// SIMATIC S7-200 project (STEP 7-Micro/WIN), CPU 226 REL 01.23

ORGANIZATION_BLOCK 主程序:OB1
TITLE=
BEGIN
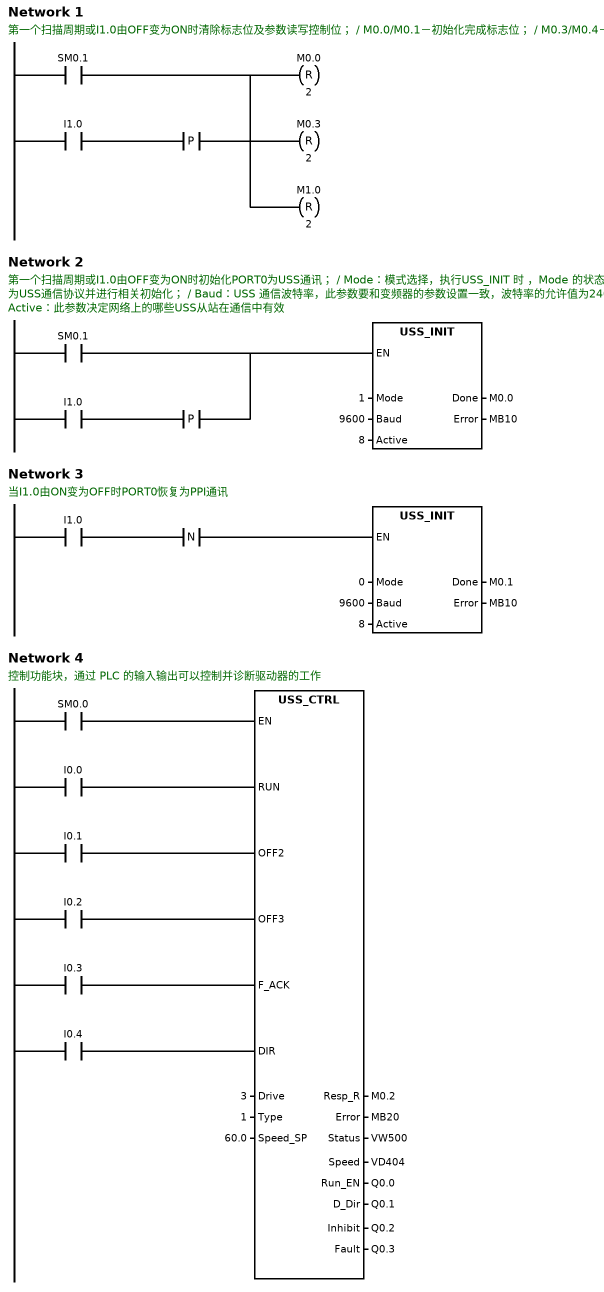
Network 1
// 第一个扫描周期或I1.0由OFF变为ON时清除标志位及参数读写控制位；
// M0.0/M0.1－初始化完成标志位；
// M0.3/M0.4－读写功能块完成标志位，用于功能块轮替；
// M1.0/M1.1－读写功能块控制位
LD     SM0.1
LD     I1.0
EU
OLD
R      M0.0, 2
R      M0.3, 2
R      M1.0, 2
Network 2
// 第一个扫描周期或I1.0由OFF变为ON时初始化PORT0为USS通讯；
// Mode：模式选择，执行USS_INIT 时 ，Mode 的状态决定 是否在Port上使用USS通信功能，0 - 恢复 Port 0 为PPI从站模式，1 - 设置 Port 0 为USS通信协议并进行相关初始化；
// Baud：USS 通信波特率，此参数要和变频器的参数设置一致，波特率的允许值为2400、4800、9600、19200、38400、57600 或115200 bit/s； 
// Active：此参数决定网络上的哪些USS从站在通信中有效
LD     SM0.1
LD     I1.0
EU
OLD
CALL   USS_INIT:SBR5, 1, 9600, 8, M0.0, MB10
Network 3
// 当I1.0由ON变为OFF时PORT0恢复为PPI通讯
LD     I1.0
ED
CALL   USS_INIT:SBR5, 0, 9600, 8, M0.1, MB10
Network 4
// 控制功能块，通过 PLC 的输入输出可以控制并诊断驱动器的工作
LD     SM0.0
=      L60.0
LD     I0.0
=      L63.7
LD     I0.1
=      L63.6
LD     I0.2
=      L63.5
LD     I0.3
=      L63.4
LD     I0.4
=      L63.3
LD     L60.0
CALL   USS_CTRL:SBR2, L63.7, L63.6, L63.5, L63.4, L63.3, 3, 1, 60.0, M0.2, MB20, VW500, VD404, Q0.0, Q0.1, Q0.2, Q0.3
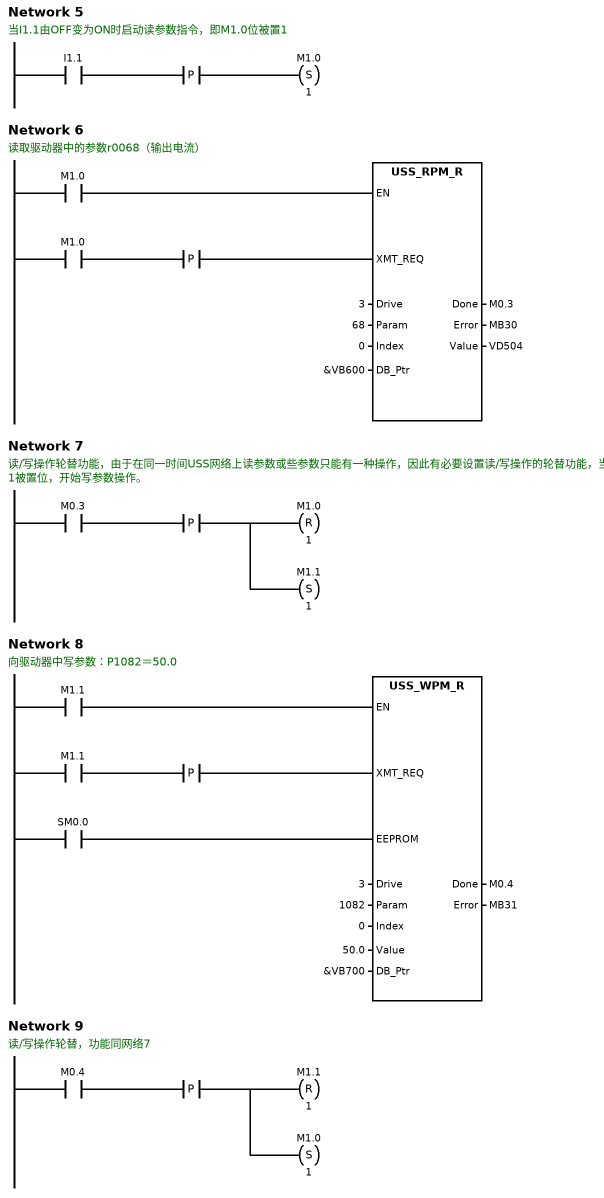
Network 5
// 当I1.1由OFF变为ON时启动读参数指令，即M1.0位被置1
LD     I1.1
EU
S      M1.0, 1
Network 6
// 读取驱动器中的参数r0068（输出电流）
LD     M1.0
=      L60.0
LD     M1.0
EU
=      L63.7
LD     L60.0
CALL   USS_RPM_R:SBR7, L63.7, 3, 68, 0, &VB600, M0.3, MB30, VD504
Network 7
// 读/写操作轮替功能，由于在同一时间USS网络上读参数或些参数只能有一种操作，因此有必要设置读/写操作的轮替功能，当读参数完成时M0.3被置1一个扫描周期，从而M1.0复位为0，读参数操作被屏蔽，同时M1.1被置位，开始写参数操作。
LD     M0.3
EU
R      M1.0, 1
S      M1.1, 1
Network 8
// 向驱动器中写参数：P1082＝50.0
LD     M1.1
=      L60.0
LD     M1.1
EU
=      L63.7
LD     SM0.0
=      L63.6
LD     L60.0
CALL   USS_WPM_R:SBR12, L63.7, L63.6, 3, 1082, 0, 50.0, &VB700, M0.4, MB31
Network 9
// 读/写操作轮替，功能同网络7
LD     M0.4
EU
R      M1.1, 1
S      M1.0, 1
END_ORGANIZATION_BLOCK

// SBR1: protected block, not included

// SBR2: protected block, not included

// SBR3: protected block, not included

// SBR4: protected block, not included

// SBR5: protected block, not included

// SBR6: protected block, not included

// SBR7: protected block, not included

// SBR8: protected block, not included

// SBR9: protected block, not included

// SBR10: protected block, not included

// SBR11: protected block, not included
